// TIA Portal V16 export
// export: Created 2021-07-12T14:47:20.8491886Z, ExportSetting WithDefaults, DisplayName Totally Integrated Automation Portal, DisplayVersion V16, DisplayName TIA Portal Version Control Interface, DisplayVersion V16, DisplayName TIA Portal Openness, DisplayVersion V16, DisplayName STEP 7 Professional, DisplayVersion V16, DisplayName STEP 7 Safety, DisplayVersion V16, DisplayName WinCC Professional, DisplayVersion V16
TYPE "SimaHydTO_typeHMIConnectionVCharEditorCommand"
TITLE = SimaHydTO_typeHMIConnectionVCharEditorCommand
// HMI interface: VChar editor - Command (HMI -> PLC)
// stored: IsFailsafeCompliant false
   STRUCT
      LoadMeasuredValues : Bool;
      LoadVChar : Bool;
      VCharLoad { S7_SetPoint := 'True'} : "SimaHydTO_typeHMIConnectionVCharSelectorCommand";
      CreateNewVChar : Bool;
      ShowPreviousRow : Bool;
      ShowNextRow : Bool;
      SaveVChar : Bool;
      SaveVCharAs : Bool;
      VCharSave { S7_SetPoint := 'True'} : "SimaHydTO_typeHMIConnectionVCharSelectorCommand";
      AbortEditor : Bool;
      DeleteRow : Bool;
      AddRow : Bool;
      SortAndDisplay : Bool;
   END_STRUCT;
END_TYPE
